INTERFACE I_REAL EXTENDS I_Datatype

{warning disable C5410}
PROPERTY PUBLIC Value : REFERENCE TO REAL
{warning restore C5410}
GET
END_GET
END_PROPERTY

END_INTERFACE

(* stored: Version 1.1.0.1, ProductVersion 3.1.4024.15
   Itf I_REAL: Id {401991fb-cfdf-0727-352e-9e4a6f57401a}
   Property Value: Id {d6f0e9a4-21b9-0c3f-0756-00b3ef4ceaa0}
   Get Get: Id {1cf58fe2-0aea-0eae-3e33-11ebd873a5eb} *)
